	sErrorDescription1 := 'User Low level errorIllegal demand data was transmitted';
	sErrorDescription2 := 'Check program';
	
9143:	
	
	sErrorDescription1 := 'User Low level errorIllegal demand data was transmitted';
	sErrorDescription2 := 'Check program';
	
9144:	
	
	sErrorDescription1 := 'User Low level errorIllegal demand data was transmitted';
	sErrorDescription2 := 'Check program';
	
9145:	
	
	sErrorDescription1 := 'User Low level errorIllegal demand data was transmitted';
	sErrorDescription2 := 'Check program';
	
9146:	
	
	sErrorDescription1 := 'User Low level errorIllegal demand data was transmitted';
	sErrorDescription2 := 'Check program';
	
9147:	
	
	sErrorDescription1 := 'User Low level errorIllegal demand data was transmitted';
	sErrorDescription2 := 'Check program';
	
9148:	
	
	sErrorDescription1 := 'User Low level errorIllegal demand data was transmitted';
	sErrorDescription2 := 'Check program';
	
9149:	
	
	sErrorDescription1 := 'User Low level errorIllegal demand data was transmitted';
	sErrorDescription2 := 'Check program';
	
9150:	
	
	sErrorDescription1 := 'User Low level errorIllegal demand data was transmitted';
	sErrorDescription2 := 'Check program';
	
9151:	
	
	sErrorDescription1 := 'User Low level errorIllegal demand data was transmitted';
	sErrorDescription2 := 'Check program';
	
9152:	
	
	sErrorDescription1 := 'User Low level errorIllegal demand data was transmitted';
	sErrorDescription2 := 'Check program';
	
9153:	
	
	sErrorDescription1 := 'User Low level errorIllegal demand data was transmitted';
	sErrorDescription2 := 'Check program';
	
9154:	
	
	sErrorDescription1 := 'User Low level errorIllegal demand data was transmitted';
	sErrorDescription2 := 'Check program';
	
9155:	
	
	sErrorDescription1 := 'User Low level errorIllegal demand data was transmitted';
	sErrorDescription2 := 'Check program';
	
9156:	
	
	sErrorDescription1 := 'User Low level errorIllegal demand data was transmitted';
	sErrorDescription2 := 'Check program';
	
9157:	
	
	sErrorDescription1 := 'User Low level errorIllegal demand data was transmitted';
	sErrorDescription2 := 'Check program';
	
9158:	
	
	sErrorDescription1 := 'User Low level errorIllegal demand data was transmitted';
	sErrorDescription2 := 'Check program';
	
9159:	
	
	sErrorDescription1 := 'User Low level errorIllegal demand data was transmitted';
	sErrorDescription2 := 'Check program';
	
9160:	
	
	sErrorDescription1 := 'User Low level errorIllegal demand data was transmitted';
	sErrorDescription2 := 'Check program';
	
9161:	
	
	sErrorDescription1 := 'User Low level errorIllegal demand data was transmitted';
	sErrorDescription2 := 'Check program';
	
9162:	
	
	sErrorDescription1 := 'User Low level errorIllegal demand data was transmitted';
	sErrorDescription2 := 'Check program';
	
9163:	
	
	sErrorDescription1 := 'User Low level errorIllegal demand data was transmitted';
	sErrorDescription2 := 'Check program';
	
9164:	
	
	sErrorDescription1 := 'User Low level errorIllegal demand data was transmitted';
	sErrorDescription2 := 'Check program';
	
9165:	
	
	sErrorDescription1 := 'User Low level errorIllegal demand data was transmitted';
	sErrorDescription2 := 'Check program';
	
9166:	
	
	sErrorDescription1 := 'User Low level errorIllegal demand data was transmitted';
	sErrorDescription2 := 'Check program';
	
9167:	
	
	sErrorDescription1 := 'User Low level errorIllegal demand data was transmitted';
	sErrorDescription2 := 'Check program';
	
9168:	
	
	sErrorDescription1 := 'User Low level errorIllegal demand data was transmitted';
	sErrorDescription2 := 'Check program';
	
9169:	
	
	sErrorDescription1 := 'User Low level errorIllegal demand data was transmitted';
	sErrorDescription2 := 'Check program';
	
9170:	
	
	sErrorDescription1 := ' User Low level errorIllegal demand data was transmitted';
	sErrorDescription2 := 'Check program';
	
9171:	
	
	sErrorDescription1 := ' User Low level errorIllegal demand data was transmitted';
	sErrorDescription2 := 'Check program';
	
9172:	
	
	sErrorDescription1 := 'User Low level errorIllegal demand data was transmitted';
	sErrorDescription2 := 'Check program';
	
9173:	
	
	sErrorDescription1 := 'User Low level errorIllegal demand data was transmitted';
	sErrorDescription2 := 'Check program';
	
9174:	
	
	sErrorDescription1 := 'User Low level errorIllegal demand data was transmitted';
	sErrorDescription2 := 'Check program';
	
9175:	
	
	sErrorDescription1 := 'User Low level errorIllegal demand data was transmitted';
	sErrorDescription2 := 'Check program';
	
9176:	
	
	sErrorDescription1 := 'User Low level errorIllegal demand data was transmitted';
	sErrorDescription2 := 'Check program';
	
9177:	
	
	sErrorDescription1 := 'User Low level errorIllegal demand data was transmitted';
	sErrorDescription2 := 'Check program';
	
9178:	
	
	sErrorDescription1 := 'User Low level errorIllegal demand data was transmitted';
	sErrorDescription2 := 'Check program';
	
9179:	
	
	sErrorDescription1 := 'User Low level errorIllegal demand data was transmitted';
	sErrorDescription2 := 'Check program';
	
9180:	
	
	sErrorDescription1 := 'User Low level errorIllegal demand data was transmitted';
	sErrorDescription2 := 'Check program';
	
9181:	
	
	sErrorDescription1 := ' User Low level errorIllegal demand data was transmitted';
	sErrorDescription2 := 'Check program';
	
9182:	
	
	sErrorDescription1 := ' User Low level errorIllegal demand data was transmitted';
	sErrorDescription2 := 'Check program';
	
9183:	
	
	sErrorDescription1 := ' User Low level errorIllegal demand data was transmitted';
	sErrorDescription2 := 'Check program';
	
9184:	
	
	sErrorDescription1 := ' User Low level errorIllegal demand data was transmitted';
	sErrorDescription2 := 'Check program';
	
9185:	
	
	sErrorDescription1 := 'User Low level errorIllegal demand data was transmitted';
	sErrorDescription2 := 'Check program';
	
9186:	
	
	sErrorDescription1 := 'User Low level errorIllegal demand data was transmitted';
	sErrorDescription2 := 'Check program';
	
9187:	
	
	sErrorDescription1 := 'User Low level errorIllegal demand data was transmitted';
	sErrorDescription2 := 'Check program';
	
9188:	
	
	sErrorDescription1 := 'User Low level errorIllegal demand data was transmitted';
	sErrorDescription2 := 'Check program';
	
9189:	
	
	sErrorDescription1 := 'User Low level errorIllegal demand data was transmitted';
	sErrorDescription2 := 'Check program';
	
9190:	
	
	sErrorDescription1 := 'User Low level errorIllegal demand data was transmitted';
	sErrorDescription2 := 'Check program';
	
9191:	
	
	sErrorDescription1 := ' User Low level errorIllegal demand data was transmitted';
	sErrorDescription2 := 'Check program';
	
9192:	
	
	sErrorDescription1 := ' User Low level errorIllegal demand data was transmitted';
	sErrorDescription2 := 'Check program';
	
9193:	
	
	sErrorDescription1 := ' User Low level errorIllegal demand data was transmitted';
	sErrorDescription2 := 'Check program';
	
9194:	
	
	sErrorDescription1 := ' User Low level errorIllegal demand data was transmitted';
	sErrorDescription2 := 'Check program';
	
9195:	
	
	sErrorDescription1 := 'User Low level errorIllegal demand data was transmitted';
	sErrorDescription2 := 'Check program';
	
9196:	
	
	sErrorDescription1 := 'User Low level errorIllegal demand data was transmitted';
	sErrorDescription2 := 'Check program';
	
9197:	
	
	sErrorDescription1 := 'User Low level errorIllegal demand data was transmitted';
	sErrorDescription2 := 'Check program';
	
9198:	
	
	sErrorDescription1 := 'User Low level errorIllegal demand data was transmitted';
	sErrorDescription2 := 'Check program';
	
9199:	
	
	sErrorDescription1 := 'User Low level errorIllegal demand data was transmitted';
	sErrorDescription2 := 'Check program';




		END_CASE
END_IF
sErrorDescription1 :=CONCAT(sErrorDescription1,': ');
sErrorDescription1 :=CONCAT(sErrorDescription1,sErrorDescription2);
END_ACTION

ACTION ErrorHandling:
//Alarm_0500	500	Error	Błąd robota {0}
IF bAlarmInit THEN
    bAlarmInit := FALSE; 
	fbSourceInfo.Clear();
	fbSourceInfo.sName:=sStationName;//'Machine';
	fbSourceInfo.nId:=iStationIndex;//2700;
	// Alarm_0500	500	Error	Błąd robota {0}
    arfbAlarm[0].CreateEx(stEventEntry := TC_EVENTS.AlarmClass.Alarm_0500, bWithConfirmation:= FALSE,  ipSourceInfo:= fbSourceInfo); 
END_IF


// Opźnienie na odczytanie kodu błędu z robota
tonbStateError(IN:= (eState = E_Station.eError) OR (eState = E_Station.eResetting), PT:=T#20MS);
bStateError	:=	tonbStateError.Q;

//tonErrorDelay(IN:=bErrorRCActive, PT:=T#200MS);
(*
IF eState = E_Station.eResetting THEN
	
	bResetErrorRC					:= bReset;
	eRunningState					:= E_RobotMovState.eReadyPlace;
	bHomingDone						:= FALSE;
	udiErrorId						:= 0;
	
ELSE
*)
(*	
	//IF tonErrorDelay.Q THEN
		bError						:= bErrorRCActive AND bEnable;
	//END_IF	
	
	IF bErrorRCActive THEN
		
		eState 						:= E_Station.eError;
		bErrorNumberRequest			:= TRUE;
		nErrorNr					:= IODATA;
		
	END_IF
	
	bResetErrorRC					:= FALSE;
	
	IF bEStop AND nErrorNr = 50 THEN
		bResetErrorRC				:= TRUE;
		//bHomingDone					:= FALSE;
	END_IF	
	
	CASE nErrorNr OF
		
		0001: sErrorDescription			:= 'Fail safe error (SRVOFF)';
		0002: sErrorDescription			:= 'Fail safe error (STOP)';
		0003: sErrorDescription			:= 'The system is abnormal.';	
		0004: sErrorDescription			:= 'CPU Watch dog error';	
		0039: sErrorDescription			:= 'Door Switch Signal line is faulty.';	
		0040: sErrorDescription			:= 'Door Switch Signal is Input';
		0041: sErrorDescription			:= 'Comm. error (Remote I/O #1).';
		0042: sErrorDescription			:= 'Comm. error (Remote I/O #2).';
		0044: sErrorDescription			:= 'OP Mode key line is faulty';
		0045: sErrorDescription			:= 'Faulty Line (T/B Enable Switch).';
		0046: sErrorDescription			:= 'Faulty wiring (Enabling Device).';
		0050: sErrorDescription			:= 'EMG signal is input. (external)';	
		0051: sErrorDescription			:= 'Wiring of the external emergency stop is abnormal.';	
		0084: sErrorDescription			:= 'Fuse is broken (O/P)';	
		0086: sErrorDescription			:= 'Hand module overcurrent';	
		0087: sErrorDescription			:= 'Fuse is blown.(Brake';	
		0088: sErrorDescription			:= 'Service I/F fuse error';	
		0090: sErrorDescription			:= 'DC24V fuse is blown';
		0091: sErrorDescription			:= 'Cant access the Special signal';
		0093: sErrorDescription			:= 'Safety relay fuse is blown';
		0094: sErrorDescription			:= 'The overcurrent in the T/B line.';
		0095: sErrorDescription			:= 'Brake release switch is turning on';
		0101: sErrorDescription			:= 'Temperature in the Controller is too high';
		0102: sErrorDescription			:= 'Temperature in the Controller is too high';
		0120: sErrorDescription			:= 'Instantaneous power failure';
		0130: sErrorDescription			:= 'The initialization connection error of system remote I/O.';
		0131: sErrorDescription			:= 'Plural Ope-panel are installed.';
		0140: sErrorDescription			:= 'Fuse is blown.(Safety unit)';
		0141: sErrorDescription			:= 'Wiring error of EMGIN connector.';
		0431: sErrorDescription			:= 'Servo amplifier motor overheat';
		0432: sErrorDescription			:= 'Servo amplifier motor overheat';
		0433: sErrorDescription			:= 'Servo amplifier motor overheat';	
		0434: sErrorDescription			:= 'Servo amplifier motor overheat';		
		1011: sErrorDescription			:= 'Wykrycie kolizji';
		1012: sErrorDescription			:= 'Wykrycie kolizji';
		1013: sErrorDescription			:= 'Wykrycie kolizji';
		1014: sErrorDescription			:= 'Wykrycie kolizji';
		
	END_CASE
	
*)
IF (bEnable) THEN
	IF  arfbAlarm[0].bActive AND bReset THEN
		bServoONRC			:= FALSE;
		bResetErrorRC		:=TRUE;
		arfbAlarm[0].Clear(nTimeStamp:=0, bResetConfirmation:= FALSE);
 	END_IF	
	IF bErrorRCActive AND (bHighLevelErrorRCActive OR bLowLevelErrorRCActive) (*AND NOT bStateError*)  THEN
		bServoONRC			:= FALSE;
// 		arfbAlarm[0].ipArguments.Clear() .AddUDInt(udiHeightServoErrorNr);
// 		IF NOT arfbAlarm[0].bActive THEN	
// 			arfbAlarm[0].Raise(nTimeStamp:=0);
// 		END_IF
// 	ELSE	
// 		IF  arfbAlarm[0].bActive AND bReset THEN
// 			arfbAlarm[0].Clear(nTimeStamp:=0, bResetConfirmation:= FALSE);
// 		END_IF
		IF NOT arfbAlarm[0].bActive THEN
			bErrorNumberRequest										:= TRUE;
		END_IF
	
		IF IODATA <> 50 AND bErrorNumberRequestActive  THEN	
			
				//bError											:= TRUE;
			IF bHighLevelErrorRCActive THEN
				udiHighLevelErrorId								:= IODATA;
				sErrorDescription2 								:= UDINT_TO_STRING(udiHighLevelErrorId); 
			END_IF
			IF bLowLevelErrorRCActive THEN
				udiLowLevelErrorId								:= IODATA;
				//udiErrorId										:= 311;
				sErrorDescription2 								:= UDINT_TO_STRING(udiHighLevelErrorId); 
				//Opis błędu
			END_IF	
			
			ErrorDescription();
			arfbAlarm[0].ipArguments.Clear() .AddString(sErrorDescription1);
				
				IF NOT arfbAlarm[0].bActive THEN	
		 			arfbAlarm[0].Raise(nTimeStamp:=0);
		 		END_IF
				
				
		
		ELSIF bErrorNumberRequestActive  AND IODATA = 50 AND bEStop THEN
			
				sErrorDescription1								:= '';
				sErrorDescription2 								:= ''; 
				bError											:= FALSE;
				bResetErrorRC									:= TRUE;
		END_IF
	
	END_IF	
 	

// 	IF bErrorRCActive AND bLowLevelErrorRCActive AND NOT bStateError THEN
// 		
// 		bError											:= TRUE;
// 		bErrorNumberRequest								:= TRUE;
// 		udiLowLevelErrorId								:= IODATA;
// 		udiErrorId										:= 311;
// 		udiErrorId										:= udiLowLevelErrorId; 
	
ELSE
//	IF  arfbAlarm[0].bActive AND bReset THEN
//	//bServoONRC							:= FALSE;	
// 		arfbAlarm[0].Clear(nTimeStamp:=0, bResetConfirmation:= FALSE);
//	END_IF
	bErrorNumberRequest									:= FALSE;	
	bError												:= 	FALSE;
	sErrorDescription1									:= '';
	sErrorDescription2 									:= ''; 
		
END_IF

(*Wyświetlanie błedu na wyjściu*)
bError							:= FALSE;
FOR nAlarmNumerator := 0 TO 19 DO
	bError						:= bError OR arfbAlarm[nAlarmNumerator].bActive;
END_FOR
	

// Przejście do eError
IF (bError AND NOT bStateError AND bEStop) THEN
	eState												:= 	E_Station.eError;
END_IF

sErrorStationName 					:= sStationName;
END_ACTION

ACTION Homing:
CASE iCaseHoming OF
	0:
		iCaseRC							:= 100;
		iCaseInit						:=0;
		IF iActualCase = 100 THEN
			iCaseRC						:= 0;
			iCaseHoming					:= 10;
		END_IF
	10:
		IF iActualCase = 150 THEN
			eState						:= E_Station.eHomingDone;
			bHomingDone					:= TRUE;
		END_IF	
END_CASE
END_ACTION

ACTION Init:
tonRetryInit(IN:=(iCaseInit = 20 OR iCaseInit = 30 OR iCaseInit = 60), PT:=T#5S);
tonReadyError(IN:=(iCaseInit=0), PT:=T#30S);

CASE iCaseInit OF
	0:
		iCaseRC								:= 0;
		bOperationEnableRC					:= FALSE;
		bServoONRC							:= FALSE;
		bRunProgramRC						:= FALSE;
		bProgramResetRC						:= FALSE;
		IF bReadyRC THEN            		
			iCaseInit						:= 10;
		END_IF                      		
	10:		                        	
		bOperationEnableRC 					:= TRUE;
		IF bOperationEnableRCActive THEN
			iCaseInit						:= 30;			//25.09.2020
		END_IF
	20:
		bProgramResetRC						:= TRUE;
		IF bProgramSelectRCActive THEN
			bProgramResetRC					:= FALSE;
			iCaseInit						:= 30;
		END_IF
		IF tonRetryInit.Q THEN
			iCaseInit						:= 0;
		END_IF
		
	30: // Reset bledu od estopa
	
		bErrorNumberRequest					:= TRUE;
		
		IF bErrorNumberRequestActive  THEN
			udiErrorIdInit					:= IODATA;	
			iCaseInit						:= iCaseInit + 10;	
		END_IF
	40: //	
		IF 	udiErrorIdInit = 50 THEN
			bResetErrorRC					:= TRUE;
			bErrorNumberRequest				:= FALSE;
			iCaseInit						:= iCaseInit +10;			
		ELSE
				iCaseInit					:= 60;
		END_IF
		
	50://
		IF 	NOT bErrorRCActive THEN
			bResetErrorRC					:= FALSE;
			iCaseInit						:= iCaseInit +10;
		END_IF		
				
	60:
		bServoONRC							:= TRUE;
		IF bServoONRCActive THEN
			iCaseInit						:= 70;
		END_IF
		IF tonRetryInit.Q THEN
			iCaseInit						:= 0;
		END_IF
	70:
		bRunProgramRC						:= TRUE;
		IF bRunProgramRCActive THEN
			iCaseInit						:= 80;
		END_IF
						
	80:
		eState 				 				:= E_Station.eReady;
	
END_CASE
END_ACTION

ACTION LubricationCounter:
(*Zliczanie cykli robota*)
rtPick(CLK:=bRun, Q=>);
IF rtPick.Q THEN
	nLubricationCounter := nLubricationCounter + 1;
END_IF
END_ACTION

ACTION Maintenance:
// Trzeba zmienic ta nazwe na wymiane baterii
IF bBatteryReplacementWasMade  THEN
	
	bBatteryReplacementDone						:= TRUE;
ELSE             
                           	
	bBatteryReplacementDone						:= FALSE;	
	
END_IF

// Wymiana Smaru

IF bGreaseReplacementWasMade AND iAxisId =1 THEN
	
	bOperationEnableRC							:= TRUE;	
	bGreaseReplacementDoneAxis1					:= TRUE;

	
ELSIF bGreaseReplacementWasMade AND iAxisId =2 THEN
	
	bOperationEnableRC							:= TRUE;
	bGreaseReplacementDoneAxis2					:= TRUE;
		
	
ELSIF bGreaseReplacementWasMade AND iAxisId =3 THEN
	
	bOperationEnableRC							:= TRUE;		
	bGreaseReplacementDoneAxis3					:= TRUE;
	
ELSE
	
	bGreaseReplacementDoneAxis1					:= FALSE;	
	bGreaseReplacementDoneAxis2					:= FALSE;
	bGreaseReplacementDoneAxis3					:= FALSE;	
	
END_IF


// Wymiana paska
IF bBeltReplacementWasMade AND iAxisId = 3 THEN
	
	bOperationEnableRC							:= TRUE;		
	bBeltReplacementDoneAxis3					:= TRUE;
	
ELSIF bBeltReplacementWasMade AND iAxisId = 4 THEN
	
	bOperationEnableRC							:= TRUE;		
	bBeltReplacementDoneAxis4					:= TRUE;
	
ELSE
	
	bBeltReplacementDoneAxis3					:= FALSE;	
	bBeltReplacementDoneAxis4					:= FALSE;

END_IF


// Reset wymiany smaru 
IF bGreaseReplacementDoneAxis1 THEN
	
	bGreaseReplacementDone 						:= TRUE;
	udiIoDATARCWrite							:= 2;
	
ELSIF bGreaseReplacementDoneAxis2 THEN	
	
	bGreaseReplacementDone 						:= TRUE;
	udiIoDATARCWrite							:= 2;

ELSIF bGreaseReplacementDoneAxis3 THEN	
	
	bGreaseReplacementDone 						:= TRUE;
	udiIoDATARCWrite							:= 4;	

ELSE
	
	bGreaseReplacementDone 						:= FALSE;	
	
END_IF

// Reset wymiany paska
IF bBeltReplacementDoneAxis3 THEN
	
	bBeltReplacementDone 						:= TRUE;
	udiIoDATARCWrite							:= 4;
	
ELSIF bBeltReplacementDoneAxis4 THEN
	
	bBeltReplacementDone 						:= TRUE;
	udiIoDATARCWrite							:= 8;	
	
ELSE
	
	bBeltReplacementDone 						:= FALSE;	
	
END_IF


// Zerowanie rozkazu resetu
IF bBatteryReplenishmentFinished THEN
	
	bBatteryReplacementDone						:= FALSE;	
	bBatteryReplacementWasMade 					:= FALSE;	
	
END_IF

IF bGreaseReplenishmentFinished THEN
	
	bGreaseReplacementDone 						:= FALSE;	
	bGreaseReplacementWasMade					:= FALSE;
	
END_IF

IF bBeltReplenishmentFinished THEN
	
	bBeltReplacementDone 						:= FALSE;
	bBeltReplacementWasMade						:= FALSE;	
	
END_IF


// Wyzerowanie wartości wpisywanej do robota
IF NOT bGreaseReplacementDoneAxis1 AND NOT bGreaseReplacementDoneAxis2 AND NOT bGreaseReplacementDoneAxis3 AND NOT bBeltReplacementDoneAxis3 AND NOT bBeltReplacementDoneAxis4 THEN
	udiIoDATARCWrite							:= 0;	
END_IF
END_ACTION

ACTION ManualMovements:
// Zboacze narastajace aktywacji edytowania ofsetu
ftCapFeederRobotEditOffset(CLK:=bEditOffset);
// Zboacze opadajace aktywacji edytowania ofsetu
rtCapFeederRobotEditOffset(CLK:=bEditOffset);

//Wywoluje akcje Maintenence do resetowania czasow baterii, smarowania i wymiany paska

Maintenance();


IF ftCapFeederRobotEditOffset.Q THEN
	bComingUp											:= TRUE;
	iCaseRC												:= 0;	
	
	//? VIS.bCapFeederRobotManualPickPlace1					:= FALSE;
	//?  VIS.bCapFeederRobotManualPickPlace2					:= FALSE;
	//?  VIS.bCapFeederRobotManualPlace						:= FALSE;
	
END_IF
IF rtCapFeederRobotEditOffset.Q THEN
	bComingUp											:= TRUE;
	bManualCatch										:= NOT bCatcherCloseSensor;
END_IF


IF bComingUp THEN
	IF bEditOffset THEN
		IF bManualPick THEN
			//iCaseRC										:= 900;
			//IF iActualCase = 900 THEN
				bComingUp								:= FALSE;
			//END_IF	
// dodaje druga pozycje pobrania			
		ELSIF bManualPick2 THEN
			//iCaseRC										:= 1600;	
			//IF iActualCase = 1600 THEN
				bComingUp								:= FALSE;
		//	END_IF		
		ELSIF bManualPlace1 THEN
			iCaseRC										:= 1100;	
			IF iActualCase = 1100 THEN
				bComingUp								:= FALSE;
			END_IF	
		ELSIF bManualPlace2 THEN
			iCaseRC										:= 1300;
			//bManualCatch								:= TRUE;
			IF iActualCase = 1300 THEN
				bComingUp								:= FALSE;
			END_IF	
		END_IF	
	ELSE	
		IF iLastCaseRC = 800 THEN												// Pozycja dolna pobierania - komenda
			iCaseRC 										:= 900;
		ELSIF iActualCase = 900 THEN											// Pozycja gorna pobierania - komenda
			iCaseRC											:= 0;
		ELSIF iActualCase = 950 THEN											// Robot w pozycji gornej pobierania
			bComingUp										:= FALSE;
			bManualPick										:= FALSE;			
		ELSIF iLastCaseRC = 1500 THEN											// Pozycja dolna pobierania 2 - komenda
			iCaseRC											:= 1600;
		ELSIF iActualCase = 1600 THEN											// Pozycja gorna pobierania 2 - komenda
			iCaseRC											:= 0;
		ELSIF iActualCase = 1650 THEN											// Robot w pozycji gornej pobierania 2
			bComingUp										:= FALSE;
			bManualPick2									:= FALSE;						
		ELSIF iLastCaseRC = 1000 THEN											// Pozycja dolna odkladania - komenda
			iCaseRC											:= 1100;
		ELSIF iActualCase = 1100 THEN											// Pozycja gorna odkladania - komenda
			iCaseRC											:= 0;
		ELSIF iActualCase = 1150 THEN											// Robot w pozycji gornej odkladania
			bComingUp										:= FALSE;
			bManualPlace1									:= FALSE;
		ELSIF iLastCaseRC = 1200 THEN											// Pozycja dolna odrzutu - komenda
			iCaseRC											:= 1300;
		ELSIF iActualCase = 1300 THEN											// Pozycja gorna odrzutu - komenda
			iCaseRC											:= 0;
		ELSIF iActualCase = 1350 THEN											// Robot w pozycji gornej odrzutu 
			bComingUp										:= FALSE;
			bManualPlace2									:= FALSE;
		END_IF
	END_IF
	iCaseManual												:= 0;	
ELSE
	IF bEditOffset THEN
		IF bManualPick THEN
			iCaseRC											:= 800;				// Pozycja dolna pobierania
		ELSIF bManualPick2 THEN                        	
			iCaseRC											:= 1500;			// Pozycja dolna pobierania 2
		ELSIF bManualPlace1 THEN                        	
			iCaseRC											:= 1000;			// Pozycja dolna odkladanie etykieciarka
		ELSIF bManualPlace2 THEN                        	
			iCaseRC											:= 1200;			// Pozycja dolna odkladania odrzut
		ELSIF iActualCase > 0 THEN                      	
			iCaseRC											:= 0;
		 	bManualPick			:= FALSE;
		 	bManualPick2		:= FALSE;			
		 	bManualPlace1		:= FALSE;
			bManualPlace2		:= FALSE;		
		END_IF	
	iCaseManual												:= 0;	
	ELSE	
//	Case pobranie pojedynczego opakowania	
		IF bManualPick THEN
			CASE iCaseManual OF
				0:
					iCaseRC										:= 200;
					IF iActualCase = 200 THEN
						iCaseRC 								:= 0;
						iCaseManual								:= 10;
					END_IF
				10: 
					IF iActualCase = 250 THEN
						iCaseManual								:= 20;
					END_IF
				20:
					bManualPick									:= FALSE;
					iCaseManual									:= 0;
			END_CASE
		END_IF	
//Dodaje Case bManualPick2 do pobrania dwoch opakowan
		IF bManualPick2 THEN
			CASE iCaseManual OF
				0:
					iCaseRC										:= 1400;
					IF iActualCase = 1400 THEN
						iCaseRC 								:= 0;
						iCaseManual								:= 10;
					END_IF
				10: 
					IF iActualCase = 1450 THEN
						iCaseManual								:= 20;
					END_IF
				20:
					bManualPick2									:= FALSE;
					iCaseManual									:= 0;
			END_CASE
		END_IF		
//	Case odlozenie opakowan na etykieciarke	
		IF bManualPlace1 THEN
			CASE iCaseManual OF
				0:
					iCaseRC										:= 300;
					IF iActualCase = 300 THEN
						iCaseRC 								:= 0;
						iCaseManual								:= 10;
					END_IF
				10: 
					IF iActualCase = 350 THEN
						iCaseManual								:= 20;
					END_IF
				20:
					bManualPlace1								:= FALSE;
					iCaseManual									:= 0;
			END_CASE
		END_IF		
//	Case odlozenie opakowan na odrzut		
		IF bManualPlace2 THEN
			CASE iCaseManual OF
				0:
					iCaseRC										:= 400;
					IF iActualCase = 400 THEN
						iCaseRC 								:= 0;
						iCaseManual								:= 10;
					END_IF
				10: 
					IF iActualCase = 450 THEN
						iCaseManual								:= 20;
					END_IF
				20:
					bManualPlace2								:= FALSE;
					iCaseManual									:= 0;
			END_CASE
		END_IF
//	Case przejazd do pozycji start inkjet		
		IF bManualStartInkJetPosition THEN
			CASE iCaseManual OF
				0:
					iCaseRC										:= 500;
					IF iActualCase = 500 THEN
						iCaseRC 								:= 0;
						iCaseManual								:= 10;
					END_IF
				10: 
					IF iActualCase = 550 THEN
						iCaseManual								:= 20;
					END_IF
				20:
					bManualStartInkJetPosition					:= FALSE;
					iCaseManual									:= 0;
			END_CASE
		END_IF
//	Case przejazd do pozycji stop inkjet		
		IF bManualStopInkJetPosition THEN
			CASE iCaseManual OF
				0:
					iCaseRC										:= 600;
					IF iActualCase = 600 THEN
						iCaseRC 								:= 0;
						iCaseManual								:= 10;
					END_IF
				10: 
					IF iActualCase = 650 THEN
						iCaseManual								:= 20;
					END_IF
				20:
					bManualStopInkJetPosition					:= FALSE;
					iCaseManual									:= 0;
			END_CASE
		END_IF	
		
		IF bManualWeightPosition THEN
			CASE iCaseManual OF
				0:
					iCaseRC										:= 660;
					IF iActualCase = 660 THEN
						iCaseRC 								:= 0;
						iCaseManual								:= 10;
					END_IF
				10: 
					IF iActualCase = 670 THEN
						iCaseManual								:= 20;
					END_IF
				20:	
					iCaseRC										:= 680;
					IF iActualCase = 680 THEN
						iCaseRC 								:= 0;
						iCaseManual								:= 30;
					END_IF	
				30:
					IF iActualCase = 690 THEN
						iCaseManual								:= 40;
					END_IF	
				40:
					bManualWeightPosition						:= FALSE;
					iCaseManual									:= 0;
			END_CASE
		END_IF
		
//	Case przejazd do pozycji gotowosci		
		IF bManualReadyPosition THEN
			CASE iCaseManual OF
				0:
					iCaseRC										:= 700;
					IF iActualCase = 700 THEN
						iCaseRC 								:= 0;
						iCaseManual								:= 10;
					END_IF
				10: 
					IF iActualCase = 750 THEN
						iCaseManual								:= 20;
					END_IF
				20:
					bManualReadyPosition						:= FALSE;
					iCaseManual									:= 0;
			END_CASE
		END_IF	
	END_IF	
END_IF	

IF iCaseRC > 0 THEN
	iLastCaseRC						:= iCaseRC;
END_IF

IF iActualCase=200 OR iActualCase=300 OR iActualCase=400 OR iActualCase=500 OR iActualCase=600 OR iActualCase=700 OR iActualCase=800 OR iActualCase=900 OR iActualCase=1000 OR iActualCase=1100 OR iActualCase=1200 OR iActualCase=1300 OR 
	iActualCase=1400 OR iActualCase=1500 OR iActualCase=1600	THEN
	iBottleTransferLock				:= 2#11111111;	//		nie moge nic
ELSIF iActualCase=150 THEN                                  
	iBottleTransferLock				:= 2#11111110;	//		moge pobrac
ELSIF iActualCase=250 OR iActualCase=950 OR iActualCase=1450 OR iActualCase=1650 THEN	           
	iBottleTransferLock				:= 2#11101001;	//		moge odłozyc, odrzucic i pojechac przed inkjet		
ELSIF iActualCase=350 OR iActualCase=1150 THEN             
	iBottleTransferLock				:= 2#11110111;	//		moge jechac tylko do gotowosci
ELSIF iActualCase=450 OR iActualCase=1350 THEN             
	iBottleTransferLock				:= 2#11110111;	//	   	moge jechac tylko do gotowosci
ELSIF iActualCase=550 THEN                                 
	iBottleTransferLock				:= 2#11011111;	//		moge jechac do koniec inkjet
ELSIF iActualCase=650 THEN                                 
	iBottleTransferLock				:= 2#10101101;	//		moge odłozyc na ety, wrocic przed inkjet
ELSIF iActualCase=750 THEN                                 
	iBottleTransferLock				:= 2#11111110;	//		moge pobrac
END_IF


(*200 pobranie opakowania, 300 odlozenie opakowania, 400 odrzucenie opakowania, 500 przejazd start inkjet, 600 przejazd stop inket, 700 powrot do gotowosci,
800 pozycja dolna pobierania manual, 900 pozycja gorna pobierana manual, 1000 Pozycja dolna odkladania - TRYB MANUALNY, 1100 Pozycja gorna odkladania - TRYB MANUALNY,
1200 Pozycja dolna odrzutu - TRYB MANUALNY, 1300 Pozycja gorna odrzutu - TRYB MANUALNY, 1400 Pobranie  2 opakowan, 1500 Pozycja dolna pobierania 2 - TRYB MANUALNY,
1600 Pozycja gorna pobierania 2 - TRYB MANUALNY


150 - koniec bazowania, 250 - koniec pobierania, 350 - koniec odkladania ety, 450 - koniec odrzutu, 550 - koniec przejazdu do start inket,
650- koniec przejazdu do stop inket, 750 - koniec przejazdu do pozycji gotowosci, 950- koniec gornej pozycji pobrania manual,
1150 - koniec górnej pozycji odkladania manual, 1350 koniec gornej pozycji odrzutu manual, 1450 - koniec pobrania dwoch opakowan,
1650 - koniec gornej pozycji pobrania manual
  *)


(*
IF iActualCase > 0 THEN
	iCaseRC										:= 0;
END_IF
*)
END_ACTION

ACTION Running:
tonWaitForSuckerSensor(IN:=(iActualCase=250 OR iActualCase=350), PT:=T#50MS);

CASE eRunningState OF
  E_RobotMovState.eReadyPlace:	
	iCaseRC								:= 0;
	IF bRun AND NOT bCycleDone THEN
		//Pobór jednego produktu
		IF iPickNumber = 1	THEN
		iCaseRC							:= 200;
			IF iActualCase = 200 THEN
				eRunningState			:= E_RobotMovState.ePicking;
			END_IF
		END_IF
		//Pobor dwóch produktów						
		IF iPickNumber = 2	THEN
		iCaseRC							:= 1400;
			IF iActualCase = 1400 THEN
				eRunningState			:= E_RobotMovState.ePicking;
			END_IF
		END_IF		
		
	END_IF
	
//Sprawdzenie czy poprawnie pobrano produkt
	
	E_RobotMovState.ePicking:
		iCaseRC							:= 0;
		IF  iActualCase = 250 OR iActualLastCase = 250 OR iActualCase = 1450 OR iActualLastCase = 1450 THEN
			iActualLastCase 			:= 0;
			eRunningState				:= E_RobotMovState.ePicked;
		END_IF	

//Sprawdzenie czy popraniw pobrano produkt po zadziałaniu estop	
	E_RobotMovState.ePickingAfterEStop:
		iCaseRC							:= 0;
		IF iActualCase = 280 OR iActualCase = 1480 THEN
			eRunningState				:= E_RobotMovState.ePicked;
		END_IF	
		
// Produkt chwycona do odłożenia 		
	E_RobotMovState.ePicked:
		IF bPlace THEN
			//Odkładanie na etykieciarke
			IF iPlaceNumber = 1 THEN
				IF bInkJetEnable THEN
					iCaseRC				:= 500;
					IF iActualCase = 500 THEN
						eRunningState	:= eMovingInkJetStartPositon;
					END_IF
				ELSE
					iCaseRC				:= 300;
					IF iActualCase = 300 THEN
						eRunningState	:= E_RobotMovState.ePlacing;
					END_IF
				END_IF	
			END_IF
			
			// Odkładanie na odrzut			
			IF iPlaceNumber = 2 THEN
				iCaseRC					:= 400;
				IF iActualCase = 400 THEN
					eRunningState		:= E_RobotMovState.eRejecting;
				END_IF
			END_IF
			
			//Przenoszenie na wagę			
			IF iPlaceNumber = 3 THEN 
				IF bInkJetEnable THEN 
					iCaseRC				:= 500;
					IF iActualCase = 500 THEN
						eRunningState	:= eMovingInkJetStartPositon;
					END_IF
				ELSE
					iCaseRC				:= 660;
					IF iActualCase = 660 THEN
						eRunningState	:= E_RobotMovState.eMovingWeightPosition;
					END_IF
				END_IF	
			END_IF	
			
			
			//Przenoszenie z obrotem
			IF iPlaceNumber = 4 THEN 
				IF bInkJetEnable THEN 
					iCaseRC				:= 500;
					IF iActualCase = 500 THEN
						eRunningState	:= eMovingInkJetStartPositon;
					END_IF
				ELSE
					iCaseRC				:= 1700;
					IF iActualCase = 1700 THEN
						eRunningState	:= E_RobotMovState.eMovingRotatedToPlace;
					END_IF
				END_IF	
			END_IF	
		END_IF		
		
// Sprawdzenie czy odłożono produkt		
	E_RobotMovState.ePlacing:	
		iCaseRC							:= 0;	
		IF iActualCase = 350 THEN
			eRunningState				:= E_RobotMovState.ePlaced;
		END_IF		
		
// Powrót do pozycji gotowości		
	E_RobotMovState.ePlaced:
		iCaseRC							:= 700;
		IF iActualCase = 700 THEN
			eRunningState				:= E_RobotMovState.eReturnToReadyPlace;
		END_IF
		
// Sprawdzenie czy odrzucono produkt		
	E_RobotMovState.eRejecting:
		iCaseRC							:= 0;
		IF iActualCase = 450 THEN	
			eRunningState				:= E_RobotMovState.eRejected;
		END_IF
		
// Sprawdzenie czy odłożono produkt na transporter odrzuconych produktów		
	E_RobotMovState.eRejected:	
		iCaseRC							:= 700;
		IF iActualCase = 700 THEN
			eRunningState				:= E_RobotMovState.eReturnToReadyPlace;
		END_IF
		
// Przejscie do pozycji poczatkowej INKJET		
	E_RobotMovState.eMovingInkJetStartPositon:
		iCaseRC							:= 0;
		IF iActualCase	= 550 THEN
			eRunningState				:= E_RobotMovState.eMovedInkJetStartPositon;
		END_IF
		
// Przejazd INKJET		
	E_RobotMovState.eMovedInkJetStartPositon:
		iCaseRC							:= 600;
		IF iActualCase = 600 THEN
			eRunningState				:= E_RobotMovState.eMovingInkJetStopPositon;
		END_IF	

// Konczenie INJET	
	E_RobotMovState.eMovingInkJetStopPositon:
		iCaseRC							:= 0;	
		IF iActualCase	= 650 THEN
			eRunningState				:= E_RobotMovState.eMovedInkJetStopPositon;
		END_IF	

// Odłożenie opakowania	
	E_RobotMovState.eMovedInkJetStopPositon:
		IF iPlaceNumber = 3 THEN //Przenoszenie na wagę
			iCaseRC				:= 660;
			IF iActualCase = 660 THEN	
				eRunningState	:= eMovingWeightPosition;				
			END_IF 
		ELSE
			iCaseRC							:= 300;	
			IF iActualCase = 300 THEN
				eRunningState				:= E_RobotMovState.ePlacing;
			END_IF	
		END_IF	
	E_RobotMovState.eMovingWeightPosition:
		iCaseRC							:= 0;	
		IF iActualCase = 670 THEN
			eRunningState				:= E_RobotMovState.eMovedWeightPosition;
		END_IF		
	E_RobotMovState.eMovedWeightPosition:
		iCaseRC							:= 680;	
		IF iActualCase = 680 THEN
			eRunningState				:= E_RobotMovState.eMovingAfterWeightPosition;
		END_IF		
	E_RobotMovState.eMovingAfterWeightPosition:
		iCaseRC							:= 0;	
		IF iActualCase = 690 THEN
			eRunningState				:= E_RobotMovState.eMovedAfterWeightPosition;
		END_IF		
	E_RobotMovState.eMovedAfterWeightPosition:
		iCaseRC							:= 300;	
		IF iActualCase = 300 THEN
			eRunningState				:= E_RobotMovState.ePlacing;
		END_IF	
//Odkładanie z obrotem		
	E_RobotMovState.eMovingRotatedToPlace:
		iCaseRC							:= 0;	
		IF iActualCase = 1750 THEN
			eRunningState				:= E_RobotMovState.eReturnToReadyPlace;
		END_IF	
//	E_RobotMovState.eMovedRoatedToPlace:
//		iCaseRC							:= 700;	
//		IF iActualCase = 700 THEN
//			eRunningState				:= E_RobotMovState.eReturnToReadyPlace;
//		END_IF	
		
	
// Konczenie cyklu	
	E_RobotMovState.eReturnToReadyPlace:	
		iCaseRC							:= 0;
		bPlace							:= FALSE;
			//IF iActualCase = 750 THEN
				iLastPickNumber			:= iPlaceNumber;
				bCycleDone				:= TRUE;
			//END_IF
END_CASE

//Tryb wolnych ruchów

IF iPlaceNumber = 1 THEN
	bSlowMotion							:= FALSE;
ELSIF iPlaceNumber = 2 THEN
	bSlowMotion							:= TRUE;	
END_IF
END_ACTION

ACTION Warning:
IF (bEnable) THEN
	
	IF bWarningAcknowledge AND bWarningRCActive  THEN
		bResetWarningRC									:= TRUE;		
	END_IF




	IF bWarningRCActive THEN
		
		bWarning										:= TRUE;
		bWarningNumberRequest							:= TRUE;
		udiWarningId									:= IODATA;
		
		CASE udiWarningId OF	
			
0013:	
	
	sWarningDescription1 := 'Illeagal fileFile Crash';
	sWarningDescription2 := 'File Initial operation';
	
0018:	
	
	sWarningDescription1 := 'The robot model was selected.The robot model was selected.';
	sWarningDescription2 := 'Reset the error';
	
0023:	
	
	sWarningDescription1 := ' Variables save failure (ProgrPower was shutdown before saving program external variables';
	sWarningDescription2 := 'It is necessary to change some parts when not improvement';
	
0024:	
	
	sWarningDescription1 := ' Variables save failure (User)Power was shutdown before saving user-defined external variables';
	sWarningDescription2 := 'The power supply unit might be deteriorated';
	
0029:	
	
	sWarningDescription1 := ' Memory error (ECC)1bit error of ECC was detected';
	sWarningDescription2 := 'When it frequently occurs, contact your service provider';
	
0102:	
	
	sWarningDescription1 := 'Temperature in the Controlle FAN check or Filter at the bottom on Controller becomes old';
	sWarningDescription2 := 'Please exchange the filter to new filter or clean up the filter';
	
0105:	
	
	sWarningDescription1 := ' Temp. in robot CPU is too higAmbient temperature of robot CPU becomes high';
	sWarningDescription2 := 'Please lower ambient temperature to the specification range';
	
0111:	
	
	sWarningDescription1 := ' No UPS battery voltageThe UPS battery is spent';
	sWarningDescription2 := 'Replace the UPS battery';
	
0112:	
	
	sWarningDescription1 := ' Open the UPS battery coverOpen the UPS battery cover';
	sWarningDescription2 := 'Close the UPS battery cover';
	
0114:	
	
	sWarningDescription1 := ' Occur the UPS warningSome abnormalities occurs in UPS';
	sWarningDescription2 := 'Please call S.C.';
	
0120:	
	
	sWarningDescription1 := 'Instantaneous power failureThe power was OFF for 20msec or more';
	sWarningDescription2 := 'Check the power supply connection and power supply state';
	
0150:	
	
	sWarningDescription1 := 'Undefined robot serial numberUndefined robot serial number';
	sWarningDescription2 := 'Input the robot serial number';
	
0151:	
	
	sWarningDescription1 := ' Undefined robot serial numberUndefined robot serial number';
	sWarningDescription2 := 'Input the robot serial number';
	
0152:	
	
	sWarningDescription1 := ' Unmatched robot serial numberRobot arm that connection was replaced';
	sWarningDescription2 := 'Please confirm the connected robot body is not replaced';
	
0190:	
	
	sWarningDescription1 := ' TB not apply present tool No.Connecting TB does not apply present tool number';
	sWarningDescription2 := 'Please operate TB after confirming present tool data(MEXTL)';
	
0200:	
	
	sWarningDescription1 := ' Err.definition file is illegaError number overlapps.';
	sWarningDescription2 := 'Correct Error definition file.';
	
0201:	
	
	sWarningDescription1 := ' Err.definition file is illegaError number is illegal.';
	sWarningDescription2 := 'Correct Error definition file.';
	
0202:	
	
	sWarningDescription1 := ' Err.definition file is illegaError number is out of the range';
	sWarningDescription2 := 'Correct Error definition file.';
	
0203:	
	
	sWarningDescription1 := ' Err.definition file is illegaError definition files form is illegal.';
	sWarningDescription2 := 'Correct Error definition file.';
	
0204:	
	
	sWarningDescription1 := ' Illegal link table was used.System Problem';
	sWarningDescription2 := 'Turn the power OFF and ON once. When it comes back, contact to the dealer.';
	
0205:	
	
	sWarningDescription1 := ' Illegal Error No.System Problem';
	sWarningDescription2 := 'Turn the power OFF and ON once. When it comes back, contact to the dealer.';
	
0240:	
	
	sWarningDescription1 := ' Setting mismatch of safety fuValid/invalid setting of the safety function is a mismatch';
	sWarningDescription2 := 'Turn the power OFF and ON once';
	
0302:	
	
	sWarningDescription1 := ' CR800 test CautionGeneral-purpose Caution for the function test of CR800';
	sWarningDescription2 := 'Check the embedded message';
	
0430:	
	
	sWarningDescription1 := ' Servo amplifier motor overheaThe motor or detectors thermal protector activated';
	sWarningDescription2 := 'Reduce the speed and acceleration of the robot';
	
0460:	
	
	sWarningDescription1 := ' Motor thermal error(Add.Axis)Overheating of the addition axis motor was detected';
	sWarningDescription2 := 'Please exchange the cooling fan of the addition axis motor';
	
1260:	
	
	sWarningDescription1 := 'Encoder communication errorInitial communication error with absolute position linear scale';
	sWarningDescription2 := 'Check the encoder cable connection and conductivity';
	
1270:	
	
	sWarningDescription1 := 'Encoder communication errorThe absolute position serial data was not transmitted correctly';
	sWarningDescription2 := 'Check the encoder cable connection and conductivity';
	
1280:	
	
	sWarningDescription1 := 'Encoder serial format errorAn error was found in the absolute position serial data format';
	sWarningDescription2 := 'Check the encoder cable connection and conductivity';
	
1290:	
	
	sWarningDescription1 := 'Absolute position fluctuationThe absolute position data fluctuated when the power ON';
	sWarningDescription2 := 'Check the axis movement due to arm dropping or external force';
	
1300:	
	
	sWarningDescription1 := 'Servo AMP MP scale F/B errorDeviation was detected in the encoder and MP scale F/B amount';
	sWarningDescription2 := 'Turn the power OFF and ON once';
	
1310:	
	
	sWarningDescription1 := 'Servo AMP MP scale offset errError in the offset data for the ABS position detection system';
	sWarningDescription2 := 'Turn the power OFF and ON once';
	
1320:	
	
	sWarningDescription1 := 'Multi-rotation data errorError was detected in the multi-rotation data for the encoder';
	sWarningDescription2 := 'Turn the power OFF and ON once';
	
1330:	
	
	sWarningDescription1 := 'Encoder battery voltage lowThe voltage of the battery supplying to the encoder has dropped';
	sWarningDescription2 := 'Replace the backup battery';
	
1340:	
	
	sWarningDescription1 := 'Over-regeneration warningThe regeneration level reached 80％ or more';
	sWarningDescription2 := 'Check the load weight or parameter SVPTYP';
	
1350:	
	
	sWarningDescription1 := 'Overload warningThe overload level of servo amplifier reached 80% or more';
	sWarningDescription2 := 'Check the load weight and the robot for collisions, etc';
	
1370:	
	
	sWarningDescription1 := 'Illegal parameter (servo)A parameter was set exceeding the setting range';
	sWarningDescription2 := 'The parameter has not been changed. Reset the correct value';
	
1400:	
	
	sWarningDescription1 := ' regeneration(AUX) frequency oRegeneration at the limit has occurred frequently';
	sWarningDescription2 := 'Check the regeneration capacity';
	
1420:	
	
	sWarningDescription1 := 'Over-regeneration warningThe overload level of converter reached 80% or more';
	sWarningDescription2 := 'Check the load weight or program';
	
1430:	
	
	sWarningDescription1 := 'Servo amplifier main circuit The servo turned ON while the main circuit power was OFF';
	sWarningDescription2 := 'Turn the main circuit power ON';
	
1520:	
	
	sWarningDescription1 := 'Servo motor output watt overThe output wattage of the servo motor exceeded ratings';
	sWarningDescription2 := 'Lower the rotation speed of the servo motor';
	
1580:	
	
	sWarningDescription1 := 'Non-registered servo warningA non-registered servo warning';
	sWarningDescription2 := 'If the warning cannot be reset, turn the power OFF and ON';
	
1620:	
	
	sWarningDescription1 := 'Illegal robot No.The designated robot No. is illegal';
	sWarningDescription2 := 'Set the correct robot No.';
	
1630:	
	
	sWarningDescription1 := 'Cannot servo ON (during errorThe servo cannot be turned ON during a servo error';
	sWarningDescription2 := 'Reset the servo error before turning the servo ON';
	
1650:	
	
	sWarningDescription1 := 'Cannot servo ON (brake OFF)The servo cannot be turned ON when the brakes release';
	sWarningDescription2 := 'Lock the brakes for all axes before turning the servo ON';
	
1660:	
	
	sWarningDescription1 := 'Cannot servo ON (SRVON procesThe servo cannot be turned ON during the servo ON process';
	sWarningDescription2 := 'Do not turn the servo ON during a servo ON process';
	
1670:	
	
	sWarningDescription1 := 'Cannot servo ON (SRVOFF proceThe servo OFF process is being carried out';
	sWarningDescription2 := 'Do not turn the servo OFF during the servo OFF process';
	
1690:	
	
	sWarningDescription1 := 'Cannot brake operation (DEADMThe brakes cannot be released while the DEADMAN switch is OFF';
	sWarningDescription2 := 'Turn the DEADMAN switch ON before operating';
	
1700:	
	
	sWarningDescription1 := 'Cannot brake operation (EMG)The brakes cannot be released while the emergency stop is input';
	sWarningDescription2 := 'Release the emergency stop state before operating';
	
1710:	
	
	sWarningDescription1 := 'Cannot brake operation (SRVONThe brakes cannot be operated during servo ON';
	sWarningDescription2 := 'Turn the servo OFF before operating';
	
1720:	
	
	sWarningDescription1 := 'Cannot brake operation (BRK OThe brakes cannot be released during the brake release process';
	sWarningDescription2 := 'Do not release the brakes during the brake release process';
	
1730:	
	
	sWarningDescription1 := 'Cannot brake operation (BRK OThe brakes cannot be locked during the brake lock process';
	sWarningDescription2 := 'Do not lock the brakes during the brake lock process';
	
1740:	
	
	sWarningDescription1 := 'Servo parameter change failurOther parameter cannot be changed during parameter change';
	sWarningDescription2 := 'Carry out the parameter change process again';
	
1750:	
	
	sWarningDescription1 := 'Servo parameter change failurChanges of the servo parameter failed';
	sWarningDescription2 := 'Carry out the parameter change process again';
	
1760:	
	
	sWarningDescription1 := 'Illegal origin dataThe origin setting data is illegal';
	sWarningDescription2 := 'Set the correct origin data';
	
1761:	
	
	sWarningDescription1 := ' Illegal origin data in robot The origin data is illegal in robot arm';
	sWarningDescription2 := 'Setting the origin';
	
1770:	
	
	sWarningDescription1 := 'Origin setting incompleteThe origin is not set';
	sWarningDescription2 := 'Re-execute after setting the origin';
	
1780:	
	
	sWarningDescription1 := 'Cannot set origin (illegal axThe origin was not set simultaneously for the interference axis';
	sWarningDescription2 := 'Set the origin simultaneously for the interference axis';
	
1781:	
	
	sWarningDescription1 := 'Cannot set origin (SRVON)The origin was set during servo ON';
	sWarningDescription2 := 'Turn the servo OFF before setting the origin';
	
1850:	
	
	sWarningDescription1 := 'Instantaneous power failureThe power was OFF for 20msec or more';
	sWarningDescription2 := 'Check the power supply connection and power supply state';
	
1870:	
	
	sWarningDescription1 := ' Cooling fan stoppedCooling fan in the controller might be out of order';
	sWarningDescription2 := 'Please exchange the cooling fan';
	
1871:	
	
	sWarningDescription1 := 'J1 cooling fan stoppedCooling fan in the controller might be out of order';
	sWarningDescription2 := 'Please exchange the cooling fan';
	
1872:	
	
	sWarningDescription1 := 'J2 cooling fan stoppedCooling fan in the controller might be out of order';
	sWarningDescription2 := 'Please exchange the cooling fan';
	
1873:	
	
	sWarningDescription1 := 'J3 cooling fan stoppedCooling fan in the controller might be out of order';
	sWarningDescription2 := 'Please exchange the cooling fan';
	
1874:	
	
	sWarningDescription1 := 'J4 cooling fan stoppedCooling fan in the controller might be out of order';
	sWarningDescription2 := 'Please exchange the cooling fan';
	
1875:	
	
	sWarningDescription1 := 'J5 cooling fan stoppedCooling fan in the controller might be out of order';
	sWarningDescription2 := 'Please exchange the cooling fan';
	
1876:	
	
	sWarningDescription1 := 'J6 cooling fan stoppedCooling fan in the controller might be out of order';
	sWarningDescription2 := 'Please exchange the cooling fan';
	
1877:	
	
	sWarningDescription1 := 'J7 cooling fan stoppedCooling fan in the controller might be out of order';
	sWarningDescription2 := 'Please exchange the cooling fan';
	
1878:	
	
	sWarningDescription1 := 'J8 cooling fan stoppedCooling fan in the controller might be out of order';
	sWarningDescription2 := 'Please exchange the cooling fan';
	
1890:	
	
	sWarningDescription1 := ' The cooling fan of the additional axis amplifier may be out of order.';
	sWarningDescription2 := '';
	
1891:	
	
	sWarningDescription1 := 'Cooling fan low rev. (add. axCooling fan of the add. axis amp. J1 might be out of order';
	sWarningDescription2 := 'Please exchange the cooling fan';
	
1892:	
	
	sWarningDescription1 := 'Cooling fan low rev. (add. axCooling fan of the add. axis amp. J2 might be out of order';
	sWarningDescription2 := 'Please exchange the cooling fan';
	
1893:	
	
	sWarningDescription1 := 'Cooling fan low rev. (add. axCooling fan of the add. axis amp. J3 might be out of order';
	sWarningDescription2 := 'Please exchange the cooling fan';
	
1894:	
	
	sWarningDescription1 := 'Cooling fan low rev. (add. axCooling fan of the add. axis amp. J4 might be out of order';
	sWarningDescription2 := 'Please exchange the cooling fan';
	
1895:	
	
	sWarningDescription1 := 'Cooling fan low rev. (add. axCooling fan of the add. axis amp. J5 might be out of order';
	sWarningDescription2 := 'Please exchange the cooling fan';
	
1896:	
	
	sWarningDescription1 := 'Cooling fan low rev. (add. axCooling fan of the add. axis amp. J6 might be out of order';
	sWarningDescription2 := 'Please exchange the cooling fan';
	
1897:	
	
	sWarningDescription1 := 'Cooling fan low rev. (add. axCooling fan of the add. axis amp. J7 might be out of order';
	sWarningDescription2 := 'Please exchange the cooling fan';
	
1898:	
	
	sWarningDescription1 := 'Cooling fan low rev. (add. axCooling fan of the add. axis amp. J8 might be out of order';
	sWarningDescription2 := 'Please exchange the cooling fan';
	
1910:	
	
	sWarningDescription1 := 'Cooling fan stopped (amp.)The cooling fan of the servo amp. stopped';
	sWarningDescription2 := 'Confirm the rotation of the servo amp. cooling fan';
	
1920:	
	
	sWarningDescription1 := 'Cooling fan stopped (pow. supThe cooling fan of the power supply stopped';
	sWarningDescription2 := 'Confirm the rotation of the power supply cooling fan';
	
1930:	
	
	sWarningDescription1 := 'Cooling fan stopped (CPU)The cooling fan of the CPU stopped';
	sWarningDescription2 := 'Confirm the rotation of the CPU cooling fan';
	
1940:	
	
	sWarningDescription1 := 'Agitating fan stoppedThe agitating fan in the controller stopped';
	sWarningDescription2 := 'Confirm the rotation of the agitating fan';
	
1960:	
	
	sWarningDescription1 := ' Additional axis AMP warningWarning of the additional axis servo amplifier was detected';
	sWarningDescription2 := 'Please refer to the manual of servo amplifier.';
	
1970:	
	
	sWarningDescription1 := ' Agitating fan stopped (robot)The agitating fan in the robot arm stopped';
	sWarningDescription2 := 'Refer to manual (Troubleshooting)';
	
1990:	
	
	sWarningDescription1 := ' Warning of encoder data errorEncoder positional data error was detected';
	sWarningDescription2 := 'Please check the counter of encoder data error';
	
2040:	
	
	sWarningDescription1 := ' Work coordinate define failedTeaching position is not correct';
	sWarningDescription2 := 'Change the teaching position';
	
2250:	
	
	sWarningDescription1 := ' Safety function is not executSafety function cannot be executed because of origin unsetting';
	sWarningDescription2 := 'Please set the origin';
	
2710:	
	
	sWarningDescription1 := 'CMP error (displacement)The amount of displacement exceeds a regulated value';
	sWarningDescription2 := 'Please reduce displacement';
	
2721:	
	
	sWarningDescription1 := 'CMP error (J1 joint angle)CMP Command exceeds the limit of J1 joint angle';
	sWarningDescription2 := 'Change the position data or reduce displacement';
	
2722:	
	
	sWarningDescription1 := 'CMP error (J2 joint angle)CMP Command exceeds the limit of J2 joint angle';
	sWarningDescription2 := 'Change the position data or reduce displacement';
	
2723:	
	
	sWarningDescription1 := 'CMP error (J3 joint angle)CMP Command exceeds the limit of J3 joint angle';
	sWarningDescription2 := 'Change the position data or reduce displacement';
	
2724:	
	
	sWarningDescription1 := 'CMP error (J4 joint angle)CMP Command exceeds the limit of J4 joint angle';
	sWarningDescription2 := 'Change the position data or reduce displacement';
	
2725:	
	
	sWarningDescription1 := 'CMP error (J5 joint angle)CMP Command exceeds the limit of J5 joint angle';
	sWarningDescription2 := 'Change the position data or reduce displacement';
	
2726:	
	
	sWarningDescription1 := 'CMP error (J6 joint angle)CMP Command exceeds the limit of J6 joint angle';
	sWarningDescription2 := 'Change the position data or reduce displacement';
	
2727:	
	
	sWarningDescription1 := 'CMP error (J7 joint angle)CMP Command exceeds the limit of J7 joint angle';
	sWarningDescription2 := 'Change the position data or reduce displacement';
	
2728:	
	
	sWarningDescription1 := 'CMP error (J8 joint angle)CMP Command exceeds the limit of J8 joint angle';
	sWarningDescription2 := 'Change the position data or reduce displacement';
	
2731:	
	
	sWarningDescription1 := 'CMP error (J1 axis speed)CMP Command exceeds the limit of J1 axis speed';
	sWarningDescription2 := 'Change the position data or reduce the robot motion speed';
	
2732:	
	
	sWarningDescription1 := 'CMP error (J2 axis speed)CMP Command exceeds the limit of J2 axis speed';
	sWarningDescription2 := 'Change the position data or reduce the robot motion speed';
	
2733:	
	
	sWarningDescription1 := 'CMP error (J3 axis speed)CMP Command exceeds the limit of J3 axis speed';
	sWarningDescription2 := 'Change the position data or reduce the robot motion speed';
	
2734:	
	
	sWarningDescription1 := 'CMP error (J4 axis speed)CMP Command exceeds the limit of J4 axis speed';
	sWarningDescription2 := 'Change the position data or reduce the robot motion speed';
	
2735:	
	
	sWarningDescription1 := 'CMP error (J5 axis speed)CMP Command exceeds the limit of J5 axis speed';
	sWarningDescription2 := 'Change the position data or reduce the robot motion speed';
	
2736:	
	
	sWarningDescription1 := 'CMP error (J6 axis speed)CMP Command exceeds the limit of J6 axis speed';
	sWarningDescription2 := 'Change the position data or reduce the robot motion speed';
	
2737:	
	
	sWarningDescription1 := 'CMP error (J7 axis speed)CMP Command exceeds the limit of J7 axis speed';
	sWarningDescription2 := 'Change the position data or reduce the robot motion speed';
	
2738:	
	
	sWarningDescription1 := 'CMP error (J8 axis speed)CMP Command exceeds the limit of J8 axis speed';
	sWarningDescription2 := 'Change the position data or reduce the robot motion speed';
	
2740:	
	
	sWarningDescription1 := 'CMP error (coordinates conv.)CMP Command (POSE type) could not convert to JOINT type';
	sWarningDescription2 := 'Change the position data';
	
2790:	
	
	sWarningDescription1 := ' Cannot teach accurate currentForce control function or CMP command is executed';
	sWarningDescription2 := ' Repeal force control function and compliance mode';
	
3989:	
	
	sWarningDescription1 := ' The test data is undecidedThe tested log data was not decided';
	sWarningDescription2 := 'Please review the argument of the FsTBat command';
	
5610:	
	
	sWarningDescription1 := 'Cannot execute during STOP ONCannot execute during stop signal input';
	sWarningDescription2 := 'Turn the stop signal OFF';
	
5670:	
	
	sWarningDescription1 := ' Cannot execute during waitCannot execute during wait';
	sWarningDescription2 := 'Execute Program Reset';
	
5680:	
	
	sWarningDescription1 := ' Cannot execute while CMP commCannot execute while CMP command is executed';
	sWarningDescription2 := 'Repeal compliance mode (execute CMP OFF)';
	
6050:	
	
	sWarningDescription1 := 'The file cannot be openedMemory size is full';
	sWarningDescription2 := 'Reduce the memory of program size';
	
6060:	
	
	sWarningDescription1 := 'The mode is not TEACHThe mode is not TEACH';
	sWarningDescription2 := 'Carry out parameter writing in the TEACH mode';
	
6070:	
	
	sWarningDescription1 := 'The time cannot be setProgram is runing or robot is SRVON';
	sWarningDescription2 := 'Check the RUN state and that the SRVON state';
	
6080:	
	
	sWarningDescription1 := 'Com mesg is too longCom mesg is too long';
	sWarningDescription2 := 'Check the various settings(ex. Parameters)';
	
6090:	
	
	sWarningDescription1 := 'Can not power reset of robotCan not power reset of robot';
	sWarningDescription2 := 'Can not power reset of robot';
	
6500:	
	
	sWarningDescription1 := 'Not opened COM lineOPEN was not executed by the program';
	sWarningDescription2 := 'Execute OPEN in the program, and then send PRN command';
	
6900:	
	
	sWarningDescription1 := 'Pseudo-input signal modeSet with the parameters';
	sWarningDescription2 := 'When using real signals mode, return the parameter';
	
7000:	
	
	sWarningDescription1 := 'Copy source file was not founThe copy source file was not found';
	sWarningDescription2 := 'Input the correct file name';
	
7010:	
	
	sWarningDescription1 := 'Delete target file was not foThe delete target file was not found';
	sWarningDescription2 := 'Input the correct file name';
	
7020:	
	
	sWarningDescription1 := 'Rename target file was not foThe rename target file was not found';
	sWarningDescription2 := 'Input the correct file name';
	
7040:	
	
	sWarningDescription1 := 'Parameter changes prohibitedChanging this parameter is prohibited as it is dangerous';
	sWarningDescription2 := 'Contact the maker';
	
7070:	
	
	sWarningDescription1 := 'Memory area is fullMemory area is full';
	sWarningDescription2 := 'Delete any unnecessary programs or data';
	
7080:	
	
	sWarningDescription1 := 'Can not read parameterNon-existent parameter or illegal password';
	sWarningDescription2 := '1. Set the correct parameter name. 2. Set the correct password';
	
7081:	
	
	sWarningDescription1 := 'Can not write parameter・Non-existent parameter or illegal password. There are a lot of numbers of characters
							Value is out of range Value is outside the range';
	sWarningDescription2 := '1. Set the correct parameter name. 2. Set the correct password';
	
7082:	
	
	sWarningDescription1 := ' Parameter writing failureFailed in writing the parameter';
	sWarningDescription2 := 'Please confirm a set value and write the parameter again';
	
7090:	
	
	sWarningDescription1 := 'Parameter comment illgalComment illgal';
	sWarningDescription2 := 'Comment is no means.';
	
7110:	
	
	sWarningDescription1 := ' Overhaul period (servo on timThe servo on time has entered the overhaul recommendation period';
	sWarningDescription2 := 'Execution of an overhaul of a robot arm is recommended period';
	
7121:	
	
	sWarningDescription1 := ' Grease replenishment period (Grease consumption degree exceeded the warning level';
	sWarningDescription2 := 'Please replenish grease and reset consumption degree';
	
7122:	
	
	sWarningDescription1 := ' Grease replenishment period (Grease consumption degree exceeded the warning level';
	sWarningDescription2 := 'Please replenish grease and reset consumption degree';
	
7123:	
	
	sWarningDescription1 := ' Grease replenishment period (Grease consumption degree exceeded the warning level';
	sWarningDescription2 := 'Please replenish grease and reset consumption degree';
	
7124:	
	
	sWarningDescription1 := ' Grease replenishment period (Grease consumption degree exceeded the warning level';
	sWarningDescription2 := 'Please replenish grease and reset consumption degree';
	
7125:	
	
	sWarningDescription1 := ' Grease replenishment period (Grease consumption degree exceeded the warning level';
	sWarningDescription2 := 'Please replenish grease and reset consumption degree';
	
7126:	
	
	sWarningDescription1 := ' Grease replenishment period (Grease consumption degree exceeded the warning level';
	sWarningDescription2 := 'Please replenish grease and reset consumption degree';
	
7131:	
	
	sWarningDescription1 := ' Timing belt replacement perioTiming belt consumption degree exceeded the warning level';
	sWarningDescription2 := 'Please replace timing belt and reset consumption degree';
	
7132:	
	
	sWarningDescription1 := ' Timing belt replacement perioTiming belt consumption degree exceeded the warning level';
	sWarningDescription2 := 'Please replace timing belt and reset consumption degree';
	
7133:	
	
	sWarningDescription1 := ' Timing belt replacement perioTiming belt consumption degree exceeded the warning level';
	sWarningDescription2 := 'Please replace timing belt and reset consumption degree';
	
7134:	
	
	sWarningDescription1 := ' Timing belt replacement perioTiming belt consumption degree exceeded the warning level';
	sWarningDescription2 := 'Please replace timing belt and reset consumption degree';
	
7135:	
	
	sWarningDescription1 := ' Timing belt replacement perioTiming belt consumption degree exceeded the warning level';
	sWarningDescription2 := 'Please replace timing belt and reset consumption degree';
	
7136:	
	
	sWarningDescription1 := ' Timing belt replacement perioTiming belt consumption degree exceeded the warning level';
	sWarningDescription2 := 'Please replace timing belt and reset consumption degree';
	
7141:	
	
	sWarningDescription1 := ' Overhaul period (decelerator)Decelerator consumption degree exceeded the warning level';
	sWarningDescription2 := 'Execution of an overhaul of a robot arm is recommended';
	
7142:	
	
	sWarningDescription1 := ' Overhaul period (decelerator)Decelerator consumption degree exceeded the warning level';
	sWarningDescription2 := 'Execution of an overhaul of a robot arm is recommended';
	
7143:	
	
	sWarningDescription1 := ' Overhaul period (decelerator)Decelerator consumption degree exceeded the warning level';
	sWarningDescription2 := 'Execution of an overhaul of a robot arm is recommended';
	
7144:	
	
	sWarningDescription1 := ' Overhaul period (decelerator)Decelerator consumption degree exceeded the warning level';
	sWarningDescription2 := 'Execution of an overhaul of a robot arm is recommended';
	
7145:	
	
	sWarningDescription1 := ' Overhaul period (decelerator)Decelerator consumption degree exceeded the warning level';
	sWarningDescription2 := 'Execution of an overhaul of a robot arm is recommended';
	
7146:	
	
	sWarningDescription1 := ' Overhaul period (decelerator)Decelerator consumption degree exceeded the warning level';
	sWarningDescription2 := 'Execution of an overhaul of a robot arm is recommended';
	
7151:	
	
	sWarningDescription1 := ' Overhaul period (bearing) (J1Bearing consumption degree exceeded the warning level';
	sWarningDescription2 := 'Execution of an overhaul of a robot arm is recommended';
	
7152:	
	
	sWarningDescription1 := ' Overhaul period (bearing) (J2Bearing consumption degree exceeded the warning level';
	sWarningDescription2 := 'Execution of an overhaul of a robot arm is recommended';
	
7153:	
	
	sWarningDescription1 := ' Overhaul period (bearing) (J3Bearing consumption degree exceeded the warning level';
	sWarningDescription2 := 'Execution of an overhaul of a robot arm is recommended';
	
7154:	
	
	sWarningDescription1 := ' Overhaul period (bearing) (J4Bearing consumption degree exceeded the warning level';
	sWarningDescription2 := 'Execution of an overhaul of a robot arm is recommended';
	
7155:	
	
	sWarningDescription1 := ' Overhaul period (bearing) (J5Bearing consumption degree exceeded the warning level';
	sWarningDescription2 := 'Execution of an overhaul of a robot arm is recommended';
	
7156:	
	
	sWarningDescription1 := ' Overhaul period (bearing) (J6Bearing consumption degree exceeded the warning level';
	sWarningDescription2 := 'Execution of an overhaul of a robot arm is recommended';
	
7161:	
	
	sWarningDescription1 := ' Overhaul period (ball screw) Ball screw consumption degree exceeded the war. level';
	sWarningDescription2 := 'Execution of an overhaul of a robot arm is recommended';
	
7162:	
	
	sWarningDescription1 := ' Overhaul period (ball screw) Ball screw consumption degree exceeded the warning level';
	sWarningDescription2 := 'Execution of an overhaul of a robot arm is recommended';
	
7163:	
	
	sWarningDescription1 := ' Overhaul period (ball screw) Ball screw consumption degree exceeded the warning level';
	sWarningDescription2 := 'Execution of an overhaul of a robot arm is recommended';
	
7164:	
	
	sWarningDescription1 := ' Overhaul period (ball screw) Ball screw consumption degree exceeded the warning level';
	sWarningDescription2 := 'Execution of an overhaul of a robot arm is recommended';
	
7165:	
	
	sWarningDescription1 := ' Overhaul period (ball screw) Ball screw consumption degree exceeded the warning level';
	sWarningDescription2 := 'Execution of an overhaul of a robot arm is recommended';
	
7166:	
	
	sWarningDescription1 := ' Overhaul period (ball screw) Ball screw consumption degree exceeded the warning level';
	sWarningDescription2 := 'Execution of an overhaul of a robot arm is recommended';
	
7170:	
	
	sWarningDescription1 := ' Abnormality detection(Dec.)The sign of failure of decelerator was detected';
	sWarningDescription2 := 'Inspection and replacement of decelerator is recommended';
	
7171:	
	
	sWarningDescription1 := ' Abnormality detection(Dec.) (The sign of failure of decelerator was detected';
	sWarningDescription2 := 'Inspection and replacement of decelerator is recommended';
	
7172:	
	
	sWarningDescription1 := ' Abnormality detection(Dec.) (The sign of failure of decelerator was detected';
	sWarningDescription2 := 'Inspection and replacement of decelerator is recommended';
	
7173:	
	
	sWarningDescription1 := ' Abnormality detection(Dec.) (The sign of failure of decelerator was detected';
	sWarningDescription2 := 'Inspection and replacement of decelerator is recommended';
	
7174:	
	
	sWarningDescription1 := ' Abnormality detection(Dec.) (The sign of failure of decelerator was detected';
	sWarningDescription2 := 'Inspection and replacement of decelerator is recommended';
	
7175:	
	
	sWarningDescription1 := ' Abnormality detection(Dec.) (The sign of failure of decelerator was detected';
	sWarningDescription2 := 'Inspection and replacement of decelerator is recommended';
	
7176:	
	
	sWarningDescription1 := ' Abnormality detection(Dec.) (The sign of failure of decelerator was detected';
	sWarningDescription2 := 'Inspection and replacement of decelerator is recommended';
	
7177:	
	
	sWarningDescription1 := ' Abnormality detection(Dec.) (The sign of failure of decelerator was detected';
	sWarningDescription2 := 'Inspection and replacement of decelerator is recommended';
	
7178:	
	
	sWarningDescription1 := ' Abnormality detection(Dec.) (The sign of failure of decelerator was detected';
	sWarningDescription2 := 'Inspection and replacement of decelerator is recommended';
	
7180:	
	
	sWarningDescription1 := ' Abnormality detection(enc datThe sign of failure of encoder was detected';
	sWarningDescription2 := 'Inspection and replacement of motor and wiring is recommended';
	
7181:	
	
	sWarningDescription1 := ' Abnormality detection(enc datThe sign of failure of encoder was detected';
	sWarningDescription2 := 'Inspection and replacement of motor and wiring is recommended';
	
7182:	
	
	sWarningDescription1 := ' Abnormality detection(enc datThe sign of failure of encoder was detected';
	sWarningDescription2 := 'Inspection and replacement of motor and wiring is recommended';
	
7183:	
	
	sWarningDescription1 := ' Abnormality detection(enc datThe sign of failure of encoder was detected';
	sWarningDescription2 := 'Inspection and replacement of motor and wiring is recommended';
	
7184:	
	
	sWarningDescription1 := ' Abnormality detection(enc datThe sign of failure of encoder was detected';
	sWarningDescription2 := 'Inspection and replacement of motor and wiring is recommended';
	
7185:	
	
	sWarningDescription1 := ' Abnormality detection(enc datThe sign of failure of encoder was detected';
	sWarningDescription2 := 'Inspection and replacement of motor and wiring is recommended';
	
7186:	
	
	sWarningDescription1 := ' Abnormality detection(enc datThe sign of failure of encoder was detected';
	sWarningDescription2 := 'Inspection and replacement of motor and wiring is recommended';
	
7187:	
	
	sWarningDescription1 := ' Abnormality detection(enc datThe sign of failure of encoder was detected';
	sWarningDescription2 := 'Inspection and replacement of motor and wiring is recommended';
	
7188:	
	
	sWarningDescription1 := ' Abnormality detection(enc datThe sign of failure of encoder was detected';
	sWarningDescription2 := 'Inspection and replacement of motor and wiring is recommended';
	
7190:	
	
	sWarningDescription1 := ' Abnormality detection(enc comThe sign of failure of encoder was detected';
	sWarningDescription2 := 'Inspection and replacement of motor and wiring is recommended';
	
7191:	
	
	sWarningDescription1 := ' Abnormality detection(enc comThe sign of failure of encoder was detected';
	sWarningDescription2 := 'Inspection and replacement of motor and wiring is recommended';
	
7192:	
	
	sWarningDescription1 := ' Abnormality detection(enc comThe sign of failure of encoder was detected';
	sWarningDescription2 := 'Inspection and replacement of motor and wiring is recommended';
	
7193:	
	
	sWarningDescription1 := ' Abnormality detection(enc comThe sign of failure of encoder was detected';
	sWarningDescription2 := 'Inspection and replacement of motor and wiring is recommended';
	
7194:	
	
	sWarningDescription1 := ' Abnormality detection(enc comThe sign of failure of encoder was detected';
	sWarningDescription2 := 'Inspection and replacement of motor and wiring is recommended';
	
7195:	
	
	sWarningDescription1 := ' Abnormality detection(enc comThe sign of failure of encoder was detected';
	sWarningDescription2 := 'Inspection and replacement of motor and wiring is recommended';
	
7196:	
	
	sWarningDescription1 := ' Abnormality detection(enc comThe sign of failure of encoder was detected';
	sWarningDescription2 := 'Inspection and replacement of motor and wiring is recommended';
	
7197:	
	
	sWarningDescription1 := ' Abnormality detection(enc comThe sign of failure of encoder was detected';
	sWarningDescription2 := 'Inspection and replacement of motor and wiring is recommended';
	
7198:	
	
	sWarningDescription1 := ' Abnormality detection(enc comThe sign of failure of encoder was detected';
	sWarningDescription2 := 'Inspection and replacement of motor and wiring is recommended';
	
7200:	
	
	sWarningDescription1 := ' Add memory has same file.Add memory has file';
	sWarningDescription2 := 'Data clear operation by TB(PROGRAM INIT)';
	
7310:	
	
	sWarningDescription1 := 'Changed variables were not save. The power was OFF during program execution';
	sWarningDescription2 := 'DO NOT turn the power OFF during PROGRAM execution';
	
7320:	
	
	sWarningDescription1 := ' Succeeded in the backup to ROBackup operation was performed';
	sWarningDescription2 := 'As it is, please use it';
	
7321:	
	
	sWarningDescription1 := ' Succeeded in the restore fromAutomatic restoration or compulsive restoration was performed';
	sWarningDescription2 := 'Since ROM data is loaded, please check the contents';
	
7322:	
	
	sWarningDescription1 := ' Failed in the backup to ROMPower supply OFF was carried out during backup processing';
	sWarningDescription2 := 'Please perform backup operation again';
	
7323:	
	
	sWarningDescription1 := ' Failed in the restore from RONone or illegal backup data. or Power supply off of processing';
	sWarningDescription2 := 'Please perform restoration operation again';
	
7324:	
	
	sWarningDescription1 := ' The capacity of ROM and RAM dThere is no extension memory for restoring';
	sWarningDescription2 := 'Please insert an extension memory correctly and perform it again';
	
7410:	
	
	sWarningDescription1 := '1 month inspection is now1 month inspection is now';
	sWarningDescription2 := '1 month inspection is now';
	
7420:	
	
	sWarningDescription1 := '3 month inspection is now3 month inspection is now';
	sWarningDescription2 := '3 month inspection is now';
	
7430:	
	
	sWarningDescription1 := '6 month inspection is now6 month inspection is now';
	sWarningDescription2 := '6 month inspection is now';
	
7440:	
	
	sWarningDescription1 := '1 year inspection is now1 year inspection is now';
	sWarningDescription2 := '1 year inspection is now';
	
7450:	
	
	sWarningDescription1 := 'No battery voltage (robot CPUThe battery is spent';
	sWarningDescription2 := 'Replace the battery and load the data';
	
7451:	
	
	sWarningDescription1 := 'Battery voltage low (robot CPThe battery is spent';
	sWarningDescription2 := 'Replace the battery';
	
7500:	
	
	sWarningDescription1 := 'No battery voltage (robot)The battery is spent';
	sWarningDescription2 := 'Replace the battery and set the origin';
	
7510:	
	
	sWarningDescription1 := 'Battery voltage low (robot)The battery is spent';
	sWarningDescription2 := 'Replace the battery';
	
7520:	
	
	sWarningDescription1 := 'Battery consumption time is oThe battery consumption time was exceeded';
	sWarningDescription2 := 'Replace the battery';
	
7530:	
	
	sWarningDescription1 := 'Replenishment time of greaseIt seems that grease reached longevity';
	sWarningDescription2 := 'Replenish grease';
	
7540:	
	
	sWarningDescription1 := 'Exchange time of the beltIt seems that the belt reached longevity';
	sWarningDescription2 := 'Execute the check and the exchange of the belt';
	
7550:	
	
	sWarningDescription1 := ' Exchange time of the deceleraIt seems that the decelerator reached longevity';
	sWarningDescription2 := 'Execute the check and the exchange of the decelerator';
	
7630:	
	
	sWarningDescription1 := ' No additional-axis cardNo additional-axis card';
	sWarningDescription2 := 'Check additional-axis card';
	
7681:	
	
	sWarningDescription1 := ' Test result was NGThe result of the test processing became NG';
	sWarningDescription2 := 'Please confirm the test object and the test condition';
	
8112:	
	
	sWarningDescription1 := ' ';
	sWarningDescription2 := '';
	
8113:	
	
	sWarningDescription1 := ' ';
	sWarningDescription2 := '';
	
8114:	
	
	sWarningDescription1 := ' ';
	sWarningDescription2 := '';
	
8115:	
	
	sWarningDescription1 := ' ';
	sWarningDescription2 := '';
	
8116:	
	
	sWarningDescription1 := ' ';
	sWarningDescription2 := '';
	
8208:	
	
	sWarningDescription1 := ' There is a possibility of theThe rewriting frequency of ROM exceeded 100000 times';
	sWarningDescription2 := 'Please do not use the trap function';
	
8490:	
	
	sWarningDescription1 := ' DEVICENET Communication test It is communication test mode';
	sWarningDescription2 := 'Please change the mode switch to 3-5 after the test ends';
	
8888:	
	
	sWarningDescription1 := ' Normal Insert-Err MsgNormal Insert-%s-Cause Msg';
	sWarningDescription2 := 'Normal Insert-%s-Measure Msg';
	
8889:	
	
	sWarningDescription1 := ' No InsertMsg-Err MsgNo InsertMsg-Cause Msg';
	sWarningDescription2 := 'No InsertMsg-Measure Msg';
	
8893:	
	
	sWarningDescription1 := ' Get Jiku Nod-Err MsgGet Jiku Nod-Cause Msg';
	sWarningDescription2 := 'Get Jiku Nod Measure Msg';
	
8921:	
	
	sWarningDescription1 := ' Caution of sensor I/F unitThe caution occurred by sensor I/F unit';
	sWarningDescription2 := 'Please refer to the manual of sensor I/F unit';
	
9200:	
	
	sWarningDescription1 := 'User Caution level errorIllegal demand data was transmitted';
	sWarningDescription2 := 'Check program';
	
9201:	
	
	sWarningDescription1 := 'User Caution level errorIllegal demand data was transmitted';
	sWarningDescription2 := 'Check program';
	
9202:	
	
	sWarningDescription1 := 'User Caution level errorIllegal demand data was transmitted';
	sWarningDescription2 := 'Check program';
	
9203:	
	
	sWarningDescription1 := 'User Caution level errorIllegal demand data was transmitted';
	sWarningDescription2 := 'Check program';
	
9204:	
	
	sWarningDescription1 := 'User Caution level errorIllegal demand data was transmitted';
	sWarningDescription2 := 'Check program';
	
9205:	
	
	sWarningDescription1 := 'User Caution level errorIllegal demand data was transmitted';
	sWarningDescription2 := 'Check program';
	
9206:	
	
	sWarningDescription1 := 'User Caution level errorIllegal demand data was transmitted';
	sWarningDescription2 := 'Check program';
	
9207:	
	
	sWarningDescription1 := 'User Caution level errorIllegal demand data was transmitted';
	sWarningDescription2 := 'Check program';
	
9208:	
	
	sWarningDescription1 := 'User Caution level errorIllegal demand data was transmitted';
	sWarningDescription2 := 'Check program';
	
9209:	
	
	sWarningDescription1 := 'User Caution level errorIllegal demand data was transmitted';
	sWarningDescription2 := 'Check program';
	
9210:	
	
	sWarningDescription1 := 'User Caution level errorIllegal demand data was transmitted';
	sWarningDescription2 := 'Check program';
	
9211:	
	
	sWarningDescription1 := 'User Caution level errorIllegal demand data was transmitted';
	sWarningDescription2 := 'Check program';
	
9212:	
	
	sWarningDescription1 := 'User Caution level errorIllegal demand data was transmitted';
	sWarningDescription2 := 'Check program';
	
9213:	
	
	sWarningDescription1 := 'User Caution level errorIllegal demand data was transmitted';
	sWarningDescription2 := 'Check program';
	
9214:	
	
	sWarningDescription1 := 'User Caution level errorIllegal demand data was transmitted';
	sWarningDescription2 := 'Check program';
	
9215:	
	
	sWarningDescription1 := 'User Caution level errorIllegal demand data was transmitted';
	sWarningDescription2 := 'Check program';
	
9216:	
	
	sWarningDescription1 := 'User Caution level errorIllegal demand data was transmitted';
	sWarningDescription2 := 'Check program';
	
9217:	
	
	sWarningDescription1 := 'User Caution level errorIllegal demand data was transmitted';
	sWarningDescription2 := 'Check program';
	
9218:	
	
	sWarningDescription1 := 'User Caution level errorIllegal demand data was transmitted';
	sWarningDescription2 := 'Check program';
	
9219:	
	
	sWarningDescription1 := 'User Caution level errorIllegal demand data was transmitted';
	sWarningDescription2 := 'Check program';
	
9220:	
	
	sWarningDescription1 := 'User Caution level errorIllegal demand data was transmitted';
	sWarningDescription2 := 'Check program';
	
9221:	
	
	sWarningDescription1 := 'User Caution level errorIllegal demand data was transmitted';
	sWarningDescription2 := 'Check program';
	
9222:	
	
	sWarningDescription1 := 'User Caution level errorIllegal demand data was transmitted';
	sWarningDescription2 := 'Check program';
	
9223:	
	
	sWarningDescription1 := 'User Caution level errorIllegal demand data was transmitted';
	sWarningDescription2 := 'Check program';
	
9224:	
	
	sWarningDescription1 := 'User Caution level errorIllegal demand data was transmitted';
	sWarningDescription2 := 'Check program';
	
9225:	
	
	sWarningDescription1 := 'User Caution level errorIllegal demand data was transmitted';
	sWarningDescription2 := 'Check program';
	
9226:	
	
	sWarningDescription1 := 'User Caution level errorIllegal demand data was transmitted';
	sWarningDescription2 := 'Check program';
	
9227:	
	
	sWarningDescription1 := 'User Caution level errorIllegal demand data was transmitted';
	sWarningDescription2 := 'Check program';
	
9228:	
	
	sWarningDescription1 := 'User Caution level errorIllegal demand data was transmitted';
	sWarningDescription2 := 'Check program';
	
9229:	
	
	sWarningDescription1 := 'User Caution level errorIllegal demand data was transmitted';
	sWarningDescription2 := 'Check program';
	
9230:	
	
	sWarningDescription1 := 'User Caution level errorIllegal demand data was transmitted';
	sWarningDescription2 := 'Check program';
	
9231:	
	
	sWarningDescription1 := 'User Caution level errorIllegal demand data was transmitted';
	sWarningDescription2 := 'Check program';
	
9232:	
	
	sWarningDescription1 := 'User Caution level errorIllegal demand data was transmitted';
	sWarningDescription2 := 'Check program';
	
9233:	
	
	sWarningDescription1 := 'User Caution level errorIllegal demand data was transmitted';
	sWarningDescription2 := 'Check program';
	
9234:	
	
	sWarningDescription1 := 'User Caution level errorIllegal demand data was transmitted';
	sWarningDescription2 := 'Check program';
	
9235:	
	
	sWarningDescription1 := 'User Caution level errorIllegal demand data was transmitted';
	sWarningDescription2 := 'Check program';
	
9236:	
	
	sWarningDescription1 := 'User Caution level errorIllegal demand data was transmitted';
	sWarningDescription2 := 'Check program';
	
9237:	
	
	sWarningDescription1 := 'User Caution level errorIllegal demand data was transmitted';
	sWarningDescription2 := 'Check program';
	
9238:	
	
	sWarningDescription1 := 'User Caution level errorIllegal demand data was transmitted';
	sWarningDescription2 := 'Check program';
	
9239:	
	
	sWarningDescription1 := 'User Caution level errorIllegal demand data was transmitted';
	sWarningDescription2 := 'Check program';
	
9240:	
	
	sWarningDescription1 := 'User Caution level errorIllegal demand data was transmitted';
	sWarningDescription2 := 'Check program';
	
9241:	
	
	sWarningDescription1 := 'User Caution level errorIllegal demand data was transmitted';
	sWarningDescription2 := 'Check program';
	
9242:	
	
	sWarningDescription1 := 'User Caution level errorIllegal demand data was transmitted';
	sWarningDescription2 := 'Check program';
	
9243:	
	
	sWarningDescription1 := 'User Caution level errorIllegal demand data was transmitted';
	sWarningDescription2 := 'Check program';
	
9244:	
	
	sWarningDescription1 := 'User Caution level errorIllegal demand data was transmitted';
	sWarningDescription2 := 'Check program';
	
9245:	
	
	sWarningDescription1 := 'User Caution level errorIllegal demand data was transmitted';
	sWarningDescription2 := 'Check program';
	
9246:	
	
	sWarningDescription1 := 'User Caution level errorIllegal demand data was transmitted';
	sWarningDescription2 := 'Check program';
	
9247:	
	
	sWarningDescription1 := 'User Caution level errorIllegal demand data was transmitted';
	sWarningDescription2 := 'Check program';
	
9248:	
	
	sWarningDescription1 := 'User Caution level errorIllegal demand data was transmitted';
	sWarningDescription2 := 'Check program';
	
9249:	
	
	sWarningDescription1 := 'User Caution level errorIllegal demand data was transmitted';
	sWarningDescription2 := 'Check program';
	
9250:	
	
	sWarningDescription1 := 'User Caution level errorIllegal demand data was transmitted';
	sWarningDescription2 := 'Check program';
	
9251:	
	
	sWarningDescription1 := 'User Caution level errorIllegal demand data was transmitted';
	sWarningDescription2 := 'Check program';
	
9252:	
	
	sWarningDescription1 := 'User Caution level errorIllegal demand data was transmitted';
	sWarningDescription2 := 'Check program';
	
9253:	
	
	sWarningDescription1 := 'User Caution level errorIllegal demand data was transmitted';
	sWarningDescription2 := 'Check program';
	
9254:	
	
	sWarningDescription1 := 'User Caution level errorIllegal demand data was transmitted';
	sWarningDescription2 := 'Check program';
	
9255:	
	
	sWarningDescription1 := 'User Caution level errorIllegal demand data was transmitted';
	sWarningDescription2 := 'Check program';
	
9256:	
	
	sWarningDescription1 := 'User Caution level errorIllegal demand data was transmitted';
	sWarningDescription2 := 'Check program';
	
9257:	
	
	sWarningDescription1 := 'User Caution level errorIllegal demand data was transmitted';
	sWarningDescription2 := 'Check program';
	
9258:	
	
	sWarningDescription1 := 'User Caution level errorIllegal demand data was transmitted';
	sWarningDescription2 := 'Check program';
	
9259:	
	
	sWarningDescription1 := 'User Caution level errorIllegal demand data was transmitted';
	sWarningDescription2 := 'Check program';
	
9260:	
	
	sWarningDescription1 := 'User Caution level errorIllegal demand data was transmitted';
	sWarningDescription2 := 'Check program';
	
9261:	
	
	sWarningDescription1 := 'User Caution level errorIllegal demand data was transmitted';
	sWarningDescription2 := 'Check program';
	
9262:	
	
	sWarningDescription1 := 'User Caution level errorIllegal demand data was transmitted';
	sWarningDescription2 := 'Check program';
	
9263:	
	
	sWarningDescription1 := 'User Caution level errorIllegal demand data was transmitted';
	sWarningDescription2 := 'Check program';
	
9264:	
	
	sWarningDescription1 := 'User Caution level errorIllegal demand data was transmitted';
	sWarningDescription2 := 'Check program';
	
9265:	
	
	sWarningDescription1 := 'User Caution level errorIllegal demand data was transmitted';
	sWarningDescription2 := 'Check program';
	
9266:	
	
	sWarningDescription1 := 'User Caution level errorIllegal demand data was transmitted';
	sWarningDescription2 := 'Check program';
	
9267:	
	
	sWarningDescription1 := 'User Caution level errorIllegal demand data was transmitted';
	sWarningDescription2 := 'Check program';
	
9268:	
	
	sWarningDescription1 := 'User Caution level errorIllegal demand data was transmitted';
	sWarningDescription2 := 'Check program';
	
9269:	
	
	sWarningDescription1 := 'User Caution level errorIllegal demand data was transmitted';
	sWarningDescription2 := 'Check program';
	
9270:	
	
	sWarningDescription1 := 'User Caution level errorIllegal demand data was transmitted';
	sWarningDescription2 := 'Check program';
	
9271:	
	
	sWarningDescription1 := 'User Caution level errorIllegal demand data was transmitted';
	sWarningDescription2 := 'Check program';
	
9272:	
	
	sWarningDescription1 := 'User Caution level errorIllegal demand data was transmitted';
	sWarningDescription2 := 'Check program';
	
9273:	
	
	sWarningDescription1 := 'User Caution level errorIllegal demand data was transmitted';
	sWarningDescription2 := 'Check program';
	
9274:	
	
	sWarningDescription1 := 'User Caution level errorIllegal demand data was transmitted';
	sWarningDescription2 := 'Check program';
	
9275:	
	
	sWarningDescription1 := 'User Caution level errorIllegal demand data was transmitted';
	sWarningDescription2 := 'Check program';
	
9276:	
	
	sWarningDescription1 := 'User Caution level errorIllegal demand data was transmitted';
	sWarningDescription2 := 'Check program';
	
9277:	
	
	sWarningDescription1 := 'User Caution level errorIllegal demand data was transmitted';
	sWarningDescription2 := 'Check program';
	
9278:	
	
	sWarningDescription1 := 'User Caution level errorIllegal demand data was transmitted';
	sWarningDescription2 := 'Check program';
	
9279:	
	
	sWarningDescription1 := 'User Caution level errorIllegal demand data was transmitted';
	sWarningDescription2 := 'Check program';
	
9280:	
	
	sWarningDescription1 := 'User Caution level errorIllegal demand data was transmitted';
	sWarningDescription2 := 'Check program';
	
9281:	
	
	sWarningDescription1 := 'User Caution level errorIllegal demand data was transmitted';
	sWarningDescription2 := 'Check program';
	
9282:	
	
	sWarningDescription1 := 'User Caution level errorIllegal demand data was transmitted';
	sWarningDescription2 := 'Check program';
	
9283:	
	
	sWarningDescription1 := 'User Caution level errorIllegal demand data was transmitted';
	sWarningDescription2 := 'Check program';
	
9284:	
	
	sWarningDescription1 := 'User Caution level errorIllegal demand data was transmitted';
	sWarningDescription2 := 'Check program';
	
9285:	
	
	sWarningDescription1 := 'User Caution level errorIllegal demand data was transmitted';
	sWarningDescription2 := 'Check program';
	
9286:	
	
	sWarningDescription1 := 'User Caution level errorIllegal demand data was transmitted';
	sWarningDescription2 := 'Check program';
	
9287:	
	
	sWarningDescription1 := 'User Caution level errorIllegal demand data was transmitted';
	sWarningDescription2 := 'Check program';
	
9288:	
	
	sWarningDescription1 := 'User Caution level errorIllegal demand data was transmitted';
	sWarningDescription2 := 'Check program';
	
9289:	
	
	sWarningDescription1 := 'User Caution level errorIllegal demand data was transmitted';
	sWarningDescription2 := 'Check program';
	
9290:	
	
	sWarningDescription1 := 'User Caution level errorIllegal demand data was transmitted';
	sWarningDescription2 := 'Check program';
	
9291:	
	
	sWarningDescription1 := 'User Caution level errorIllegal demand data was transmitted';
	sWarningDescription2 := 'Check program';
	
9292:	
	
	sWarningDescription1 := 'User Caution level errorIllegal demand data was transmitted';
	sWarningDescription2 := 'Check program';
	
9293:	
	
	sWarningDescription1 := 'User Caution level errorIllegal demand data was transmitted';
	sWarningDescription2 := 'Check program';
	
9294:	
	
	sWarningDescription1 := 'User Caution level errorIllegal demand data was transmitted';
	sWarningDescription2 := 'Check program';
	
9295:	
	
	sWarningDescription1 := 'User Caution level errorIllegal demand data was transmitted';
	sWarningDescription2 := 'Check program';
	
9296:	
	
	sWarningDescription1 := 'User Caution level errorIllegal demand data was transmitted';
	sWarningDescription2 := 'Check program';
	
9297:	
	
	sWarningDescription1 := 'User Caution level errorIllegal demand data was transmitted';
	sWarningDescription2 := 'Check program';
	
9298:	
	
	sWarningDescription1 := 'User Caution level errorIllegal demand data was transmitted';
	sWarningDescription2 := 'Check program';
	
9299:	
	
	sWarningDescription1 := 'User Caution level errorIllegal demand data was transmitted';
	sWarningDescription2 := 'Check program';

			
		END_CASE
		
	ELSE
	bWarningNumberRequest									:= FALSE;
	bResetWarningRC											:= FALSE;	
	bWarning												:= FALSE;
	sWarningDescription1									:= '';
	sWarningDescription2 									:= ''; 
	
	END_IF
	
ELSE
	udiWarningId											:= 0;
	bWarning												:= 	FALSE;
	sWarningDescription1									:= '';
	sWarningDescription2 									:= ''; 
		
END_IF
END_ACTION

END_FUNCTION_BLOCK

(* stored: Version 1.2.0.0, ProductVersion 3.1.4026.13, FileIdentifier 70beb0e39faa415c4ee0f93c7be47a6437ab3095, FileSignature 91b9f591da5731d6bb0da43ed400bb2d26d484e2e927f42fc38e78c08067ccb17642b087e73dc520ed2e5f4572d992d65120639efe93267b68f945de6e45fc48734de02ffa2ddf474a0e1b62146173677955ac246c20ce2404337a95ec7303fff75973663d581cd9b3e223365de8fa64b0ddbb07d55efaf878028d9e597cdeda8405d63db374860f3322c933a1744afecb9387bfd87453a01817c0b3eaee6d4df6d264a59cbae6ba8a2003597d6200237288e974994cb6440402a428a70b25284d2b2f411b60feb9a1cb5c9de71077426aef72227febe1dd14c6eafdd274424c5c47aed8bbbf6adc7c454705bf787c48fd29d15b9ba4c5870d08ea7c2433490f
   POU FB_Robot2Bottles: Id {8292d546-511c-4e1d-a3b9-c60838ad1033}, SpecialFunc None
   Action aStationID: Id {41eeae34-9f1e-48c8-a23f-f9dc92796360}
   Action aStatistic: Id {214ed6b2-f089-493b-ba60-4a32ce11edab}
   Action Control: Id {1a46f924-0f1d-4f44-9b8e-2d627ae8ab03}
   Action DataExchange: Id {330ba392-f723-48e8-bda3-d98abc925b74}
   Action ErrorDescription: Id {df89e751-12e7-43ee-a2c3-6d9bcfafcdc2}
   Action ErrorHandling: Id {846d74be-d373-4763-b1de-14e2546d6156}
   Action Homing: Id {43d4f581-300e-4b16-ab06-aa76b5166d76}
   Action Init: Id {83dce899-c44a-4f21-a5ed-382309bdad5e}
   Action LubricationCounter: Id {142e8749-2056-4ffd-83ba-7a6efdf5fb74}
   Action Maintenance: Id {3e69b75e-e1ad-48a3-be57-16c4dae37ad3}
   Action ManualMovements: Id {71b218b8-e4ce-4a3f-acc2-7e353e06e163}
   Action Running: Id {3d5400bb-6c51-4314-99d1-15ad56382084}
   Action Warning: Id {81505606-a67c-452d-96a6-75ecc544df36} *)
